# EPICS autosave request: alicatGasFlow/alicatPressureCtrl_settings.req
$(P)$(Q):DGAIN:WR
$(P)$(Q):PGAIN:WR
